FUNCTION TransferChemical : BOOL
VAR_INPUT
	pTank : POINTER TO ST_Tank;
END_VAR
VAR
	
END_VAR

IF pTank <> 0 THEN
	IF pTank^.fLevel > GVL.fRequiredLevel THEN
		pTank^.fLevel := pTank^.fLevel - GVL.fTransferSpeed;
	ELSE
		PTank^.bLevelAlarm := FALSE;
	END_IF
END_IF

END_FUNCTION

(* stored: Version 1.1.0.1, ProductVersion 3.1.4024.16
   POU TransferChemical: Id {0653ac06-573f-4c7b-bf90-3d41a5ddce1e}, SpecialFunc None *)
